FUNCTION_BLOCK FB_SafetyGuard
VAR_INPUT
	shuttle_crash_detector						:BOOL;
	emergency_stop									:BOOL;
	limit_switch										:BOOL;
	interlock_triggered								:BOOL;//安全门被触发
	LightCurtainTriggered							:BOOL;
END_VAR
VAR_OUTPUT
	error_code			:INT;
	state						:INT;
	Init_Done				:BOOL;
	Error						:BOOL;
END_VAR
VAR
	step    				:INT;
	ton1					:Tc2_Standard.TON;
END_VAR
VAR_IN_OUT
	Initialize			:BOOL;
	SetOff			:BOOL;
END_VAR

CASE  step OF
0://waiting
	IF Initialize THEN 
		step:=5;
	ELSIF SetOff OR GVL.Reset THEN 
		step:=99;
	END_IF
	
	(******************状态自复位***************************)
	ton1(IN:=Init_Done  , PT:=T#1S , Q=> , ET=> );
	IF ton1.Q THEN 
		Init_Done:=FALSE;
	END_IF
5://OFF
	state:=SafetyGuardStateEnum.off;
	error_code:=SafetyGuardErrorEnum.no_error;
	
	IF Initialize THEN 
		Initialize:=FALSE;
		step:=10;
	END_IF
10://Initializing
	state:=SafetyGuardStateEnum.initializing;
	
	step:=20;
20://ready
	Init_Done:=TRUE;
	state:=SafetyGuardStateEnum.ready;
	step:=0;

99://SetOff
	SetOff:=FALSE;
	Error:=FALSE;
	state:=SafetyGuardStateEnum.off;
	error_code:=SafetyGuardErrorEnum.no_error;
	step:=0;
100://error
		state:=SafetyGuardStateEnum.error;
		Error:=TRUE;
		step:=0;
END_CASE

IF SetOff OR GVL.Reset THEN 
		step:=99;
END_IF

IF state <>SafetyGuardStateEnum.off AND state <>SafetyGuardStateEnum.error THEN 
		IF emergency_stop THEN 
		error_code:=SafetyGuardErrorEnum.emergency_error;
		step:=100;
	ELSIF 	interlock_triggered THEN 
		error_code:=SafetyGuardErrorEnum.interlock_error;
		step:=100;
	ELSIF	shuttle_crash_detector THEN 
		error_code:=SafetyGuardErrorEnum.shuttle_crash_error;
		step:=100;
	ELSIF	limit_switch THEN 
		error_code:=SafetyGuardErrorEnum.limit_switch_error;
		step:=100;
	END_IF
END_IF

END_FUNCTION_BLOCK

(* stored: Version 1.1.0.1, ProductVersion 3.1.4024.11
   POU FB_SafetyGuard: Id {79ee3705-253c-4b69-a96a-b6ceb5159aef}, SpecialFunc None *)
